TYPE ST_EventHmiControl :
STRUCT
END_STRUCT
END_TYPE

(* stored: Version 1.1.0.1, ProductVersion 3.1.4026.18
   DUT ST_EventHmiControl: Id {db9a39da-6fd4-4a29-b385-e98644c5336f} *)
